FUNCTION_BLOCK GearMover EXTENDS FB_Mover IMPLEMENTS IGearMover
VAR_INPUT
	XtsTrack : IXtsTrack;
	StateMachine : IPmlStateMachine;
END_VAR
VAR_OUTPUT
END_VAR
VAR
	moverSequence : GearMoverSequence;
	bInit : BOOL;
	CurrentLimit AT%Q* : INT;
	Mode AT%Q* : UINT;
	axesGear	: GearInCA;
	isMasterAxis: BOOL;
	MoverToGearTo: UDINT := 1;
END_VAR
VAR_IN_OUT
	MoverArray : ARRAY[*] OF IGearMover;
END_VAR

IF NOT bInit THEN
	bInit := TRUE;
	_trackLength := XtsTrack.TrackLength;
	IF (THIS^._axis.NcToPlc.AxisId MOD 2)<>1 THEN
		Mode.8 := TRUE;
		isMasterAxis := TRUE;
		CurrentLimit := 3000;
	ELSE
		isMasterAxis := FALSE;
		MoverToGearTo := THIS^.AxisRef.NcToPlc.AxisId + 1;
	END_IF
END_IF

SUPER^();
axesGear(_MasterAxis := MoverArray[MoverToGearTo].AxisRef, _SlaveAxis := THIS^.AxisRef);
moverSequence(ThisMover := THIS^,
				XtsTrack := XtsTrack,
				StateMachine := StateMachine,
				MoverArray := MoverArray);

METHOD PUBLIC Gear : BOOL
VAR_INPUT
	MasterPosition : MC_LREAL;
	SlavePosition : MC_LREAL;
END_VAR
IF NOT axesGear.Busy THEN
		axesGear.Sync(MasterPosition := MasterPosition, SlavePosition := SlavePosition);
		Gear := TRUE;
END_IF
END_METHOD

METHOD inGear : BOOL
VAR_INPUT
END_VAR
inGear := axesGear.gearInCA.InSync;
END_METHOD

METHOD isMaster : BOOL
VAR_INPUT
END_VAR
isMaster := isMasterAxis;
END_METHOD

METHOD masterAxis : UDINT
VAR_INPUT
END_VAR
masterAxis := MoverToGearTo;
END_METHOD

END_FUNCTION_BLOCK

(* stored: Version 1.1.0.1, ProductVersion 3.1.4024.9
   POU GearMover: Id {ff37142b-1aaf-40b6-8a09-27f219b6fa6d}, SpecialFunc None
   Method Gear: Id {e70c4ab6-700a-4f7f-96e2-f6bea672eae8}
   Method inGear: Id {9ee658e1-449f-4c40-a0f1-11ea83a98b8e}
   Method isMaster: Id {0b9c72f9-349e-45a4-a413-9118e25a1eb6}
   Method masterAxis: Id {9f943dc0-f377-431c-9b83-a2dfc72d5fd9} *)
